(* IEC 61131-3 sources: rep_b/Projects/Extended_block/Strategy/Task-Main, 3 files *)

(* ---- GlobalVars.st ---- *)
VAR_GLOBAL
	IsSlaveController:BOOL:=FALSE;   //delete

END_VAR

(* ---- RetainGlobalVars.st ---- *)
VAR_GLOBAL RETAIN

	SlavePCOtype:UINT;  //тип ведомого контроллера

END_VAR

(* ---- Main.st ---- *)
PROGRAM main

{REGION Inizialisation. Send to Master type of controller}

IF INIZIALIZATION_1 = FALSE THEN
	SlavePCOtype:=GET_BOARD_TYPE();
	INIZIALIZATION_1:=TRUE;
	RETURN;
END_IF;

PLAN_BOARD_TYPE:=UINT_TO_INT(SlavePCOtype);

{ENDREGION}

END_PROGRAM
